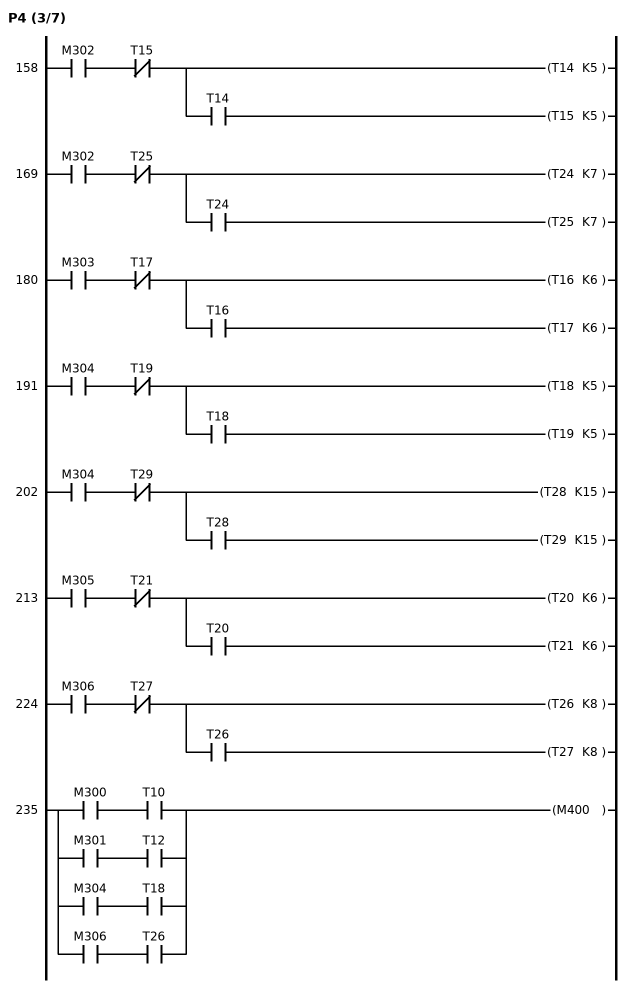
[picture p24: ladder of P4, rungs at steps 158 to 235]
158   LD      M302
      ANI     T15
      OUT     T14 K5
      AND     T14
      OUT     T15 K5
169   LD      M302
      ANI     T25
      OUT     T24 K7
      AND     T24
      OUT     T25 K7
180   LD      M303
      ANI     T17
      OUT     T16 K6
      AND     T16
      OUT     T17 K6
191   LD      M304
      ANI     T19
      OUT     T18 K5
      AND     T18
      OUT     T19 K5
202   LD      M304
      ANI     T29
      OUT     T28 K15
      AND     T28
      OUT     T29 K15
213   LD      M305
      ANI     T21
      OUT     T20 K6
      AND     T20
      OUT     T21 K6
224   LD      M306
      ANI     T27
      OUT     T26 K8
      AND     T26
      OUT     T27 K8
235   LD      M300
      AND     T10
      LD      M301
      AND     T12
      ORB
      LD      M304
      AND     T18
      ORB
      LD      M306
      AND     T26
      ORB
      OUT     M400
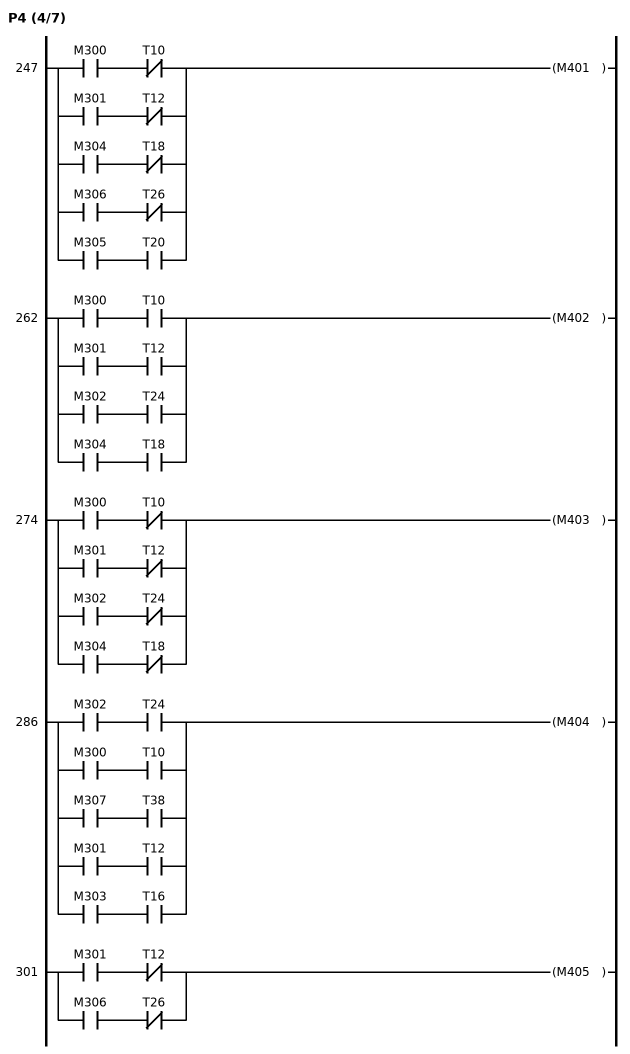
247   LD      M300
      ANI     T10
      LD      M301
      ANI     T12
      ORB
      LD      M304
      ANI     T18
      ORB
      LD      M306
      ANI     T26
      ORB
      LD      M305
      AND     T20
      ORB
      OUT     M401
262   LD      M300
      AND     T10
      LD      M301
      AND     T12
      ORB
      LD      M302
      AND     T24
      ORB
      LD      M304
      AND     T18
      ORB
      OUT     M402
274   LD      M300
      ANI     T10
      LD      M301
      ANI     T12
      ORB
      LD      M302
      ANI     T24
      ORB
      LD      M304
      ANI     T18
      ORB
      OUT     M403
286   LD      M302
      AND     T24
      LD      M300
      AND     T10
      ORB
      LD      M307
      AND     T38
      ORB
      LD      M301
      AND     T12
      ORB
      LD      M303
      AND     T16
      ORB
      OUT     M404
301   LD      M301
      ANI     T12
      LD      M306
      ANI     T26
      ORB
      OUT     M405
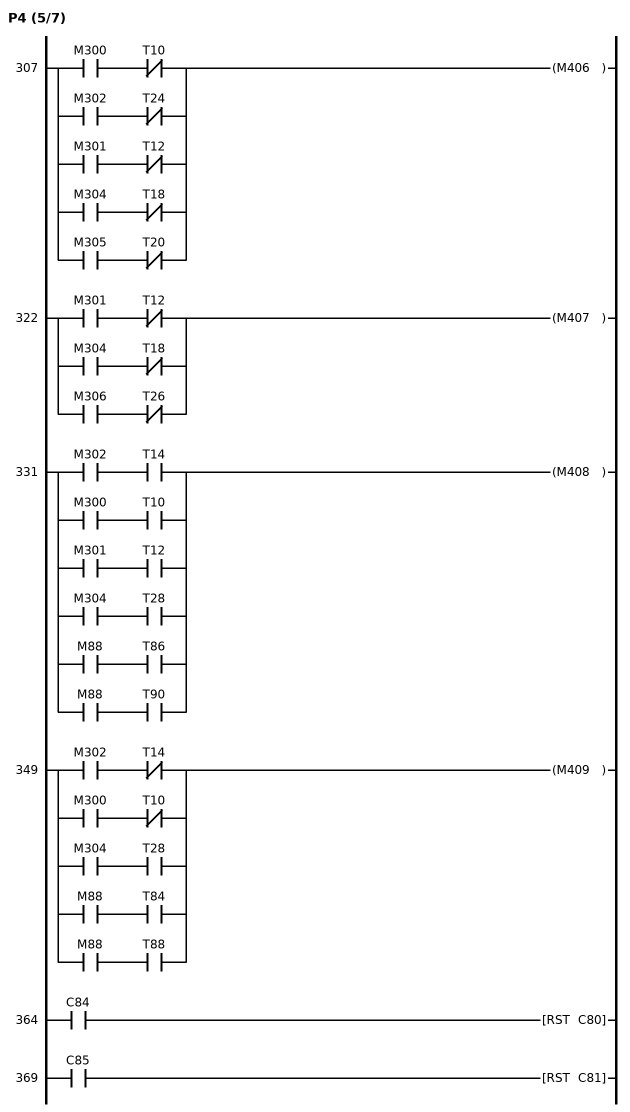
307   LD      M300
      ANI     T10
      LD      M302
      ANI     T24
      ORB
      LD      M301
      ANI     T12
      ORB
      LD      M304
      ANI     T18
      ORB
      LD      M305
      ANI     T20
      ORB
      OUT     M406
322   LD      M301
      ANI     T12
      LD      M304
      ANI     T18
      ORB
      LD      M306
      ANI     T26
      ORB
      OUT     M407
331   LD      M302
      AND     T14
      LD      M300
      AND     T10
      ORB
      LD      M301
      AND     T12
      ORB
      LD      M304
      AND     T28
      ORB
      LD      M88
      AND     T86
      ORB
      LD      M88
      AND     T90
      ORB
      OUT     M408
349   LD      M302
      ANI     T14
      LD      M300
      ANI     T10
      ORB
      LD      M304
      AND     T28
      ORB
      LD      M88
      AND     T84
      ORB
      LD      M88
      AND     T88
      ORB
      OUT     M409
364   LD      C84
      RST     C80
369   LD      C85
      RST     C81
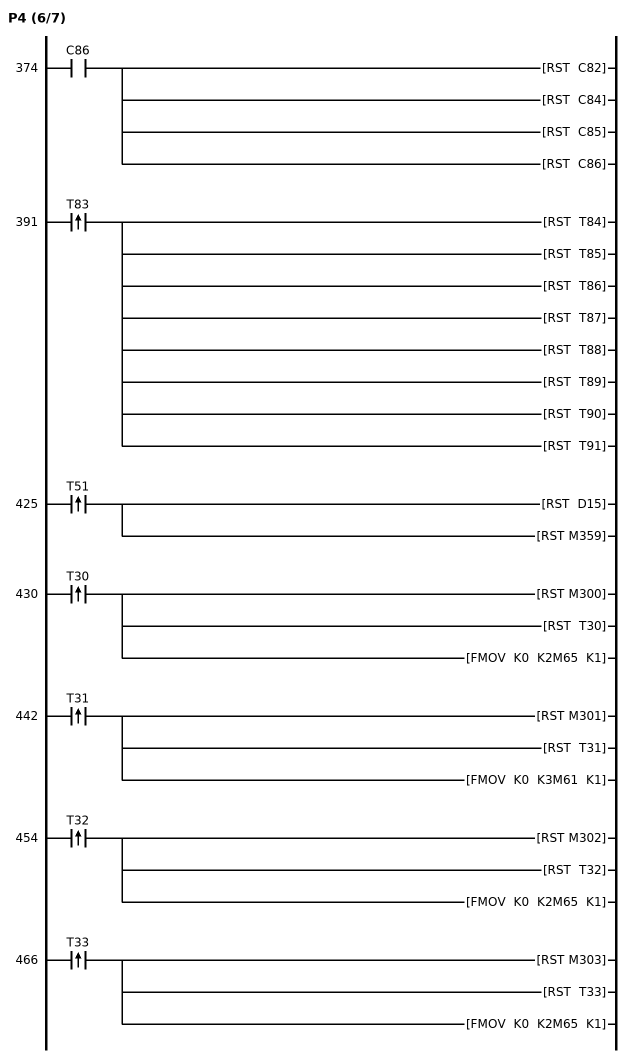
374   LD      C86
      RST     C82
      RST     C84
      RST     C85
      RST     C86
391   LDP     T83
      RST     T84
      RST     T85
      RST     T86
      RST     T87
      RST     T88
      RST     T89
      RST     T90
      RST     T91
425   LDP     T51
      RST     D15
      RST     M359
430   LDP     T30
      RST     M300
      RST     T30
      FMOV    K0 K2M65 K1
442   LDP     T31
      RST     M301
      RST     T31
      FMOV    K0 K3M61 K1
454   LDP     T32
      RST     M302
      RST     T32
      FMOV    K0 K2M65 K1
466   LDP     T33
      RST     M303
      RST     T33
      FMOV    K0 K2M65 K1
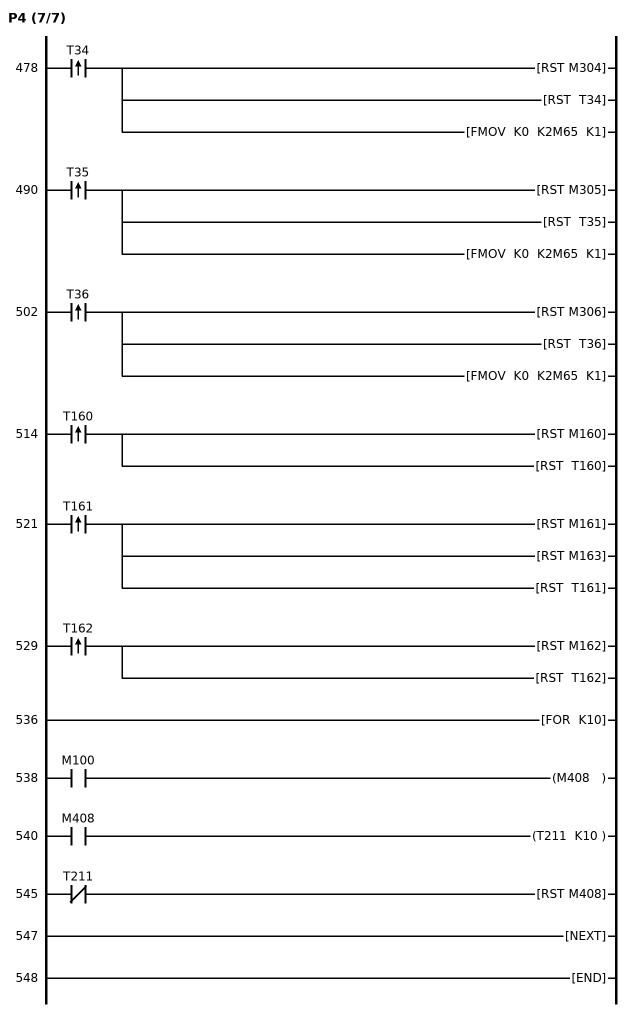
478   LDP     T34
      RST     M304
      RST     T34
      FMOV    K0 K2M65 K1
490   LDP     T35
      RST     M305
      RST     T35
      FMOV    K0 K2M65 K1
502   LDP     T36
      RST     M306
      RST     T36
      FMOV    K0 K2M65 K1
514   LDP     T160
      RST     M160
      RST     T160
521   LDP     T161
      RST     M161
      RST     M163
      RST     T161
529   LDP     T162
      RST     M162
      RST     T162
536   FOR     K10
538   LD      M100
      OUT     M408
540   LD      M408
      OUT     T211 K10
545   LDI     T211
      RST     M408
547   NEXT
548   END
END_PROGRAM

PROGRAM P5
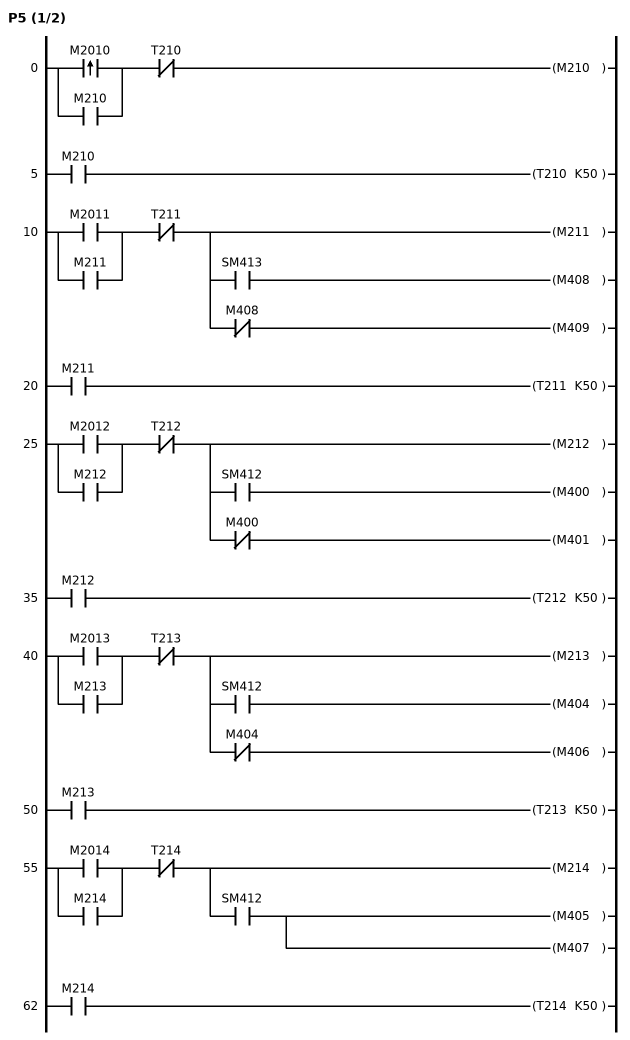
0     LDP     M2010
      OR      M210
      ANI     T210
      OUT     M210
5     LD      M210
      OUT     T210 K50
10    LD      M2011
      OR      M211
      ANI     T211
      OUT     M211
      MPS
      AND     SM413
      OUT     M408
      MPP
      ANI     M408
      OUT     M409
20    LD      M211
      OUT     T211 K50
25    LD      M2012
      OR      M212
      ANI     T212
      OUT     M212
      MPS
      AND     SM412
      OUT     M400
      MPP
      ANI     M400
      OUT     M401
35    LD      M212
      OUT     T212 K50
40    LD      M2013
      OR      M213
      ANI     T213
      OUT     M213
      MPS
      AND     SM412
      OUT     M404
      MPP
      ANI     M404
      OUT     M406
50    LD      M213
      OUT     T213 K50
55    LD      M2014
      OR      M214
      ANI     T214
      OUT     M214
      AND     SM412
      OUT     M405
      OUT     M407
62    LD      M214
      OUT     T214 K50
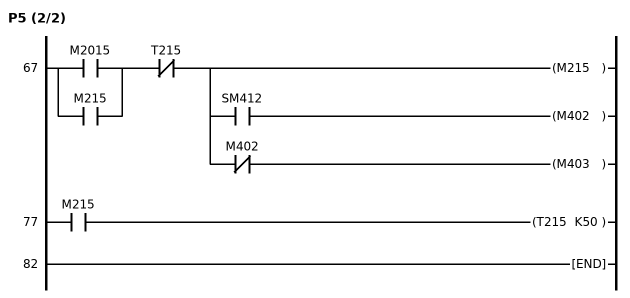
67    LD      M2015
      OR      M215
      ANI     T215
      OUT     M215
      MPS
      AND     SM412
      OUT     M402
      MPP
      ANI     M402
      OUT     M403
77    LD      M215
      OUT     T215 K50
82    END
END_PROGRAM

PROGRAM P6
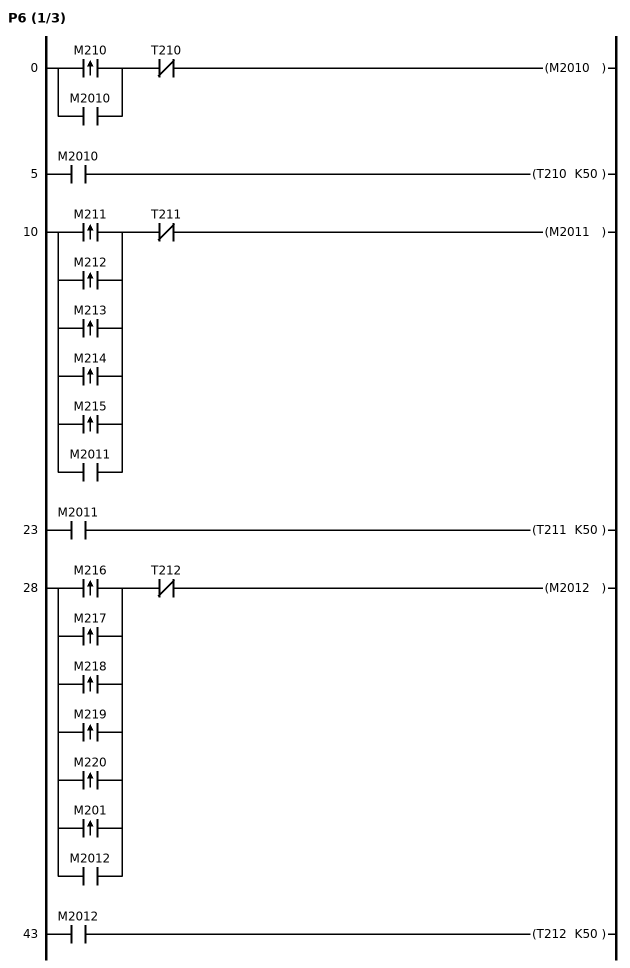
0     LDP     M210
      OR      M2010
      ANI     T210
      OUT     M2010
5     LD      M2010
      OUT     T210 K50
10    LDP     M211
      ORP     M212
      ORP     M213
      ORP     M214
      ORP     M215
      OR      M2011
      ANI     T211
      OUT     M2011
23    LD      M2011
      OUT     T211 K50
28    LDP     M216
      ORP     M217
      ORP     M218
      ORP     M219
      ORP     M220
      ORP     M201
      OR      M2012
      ANI     T212
      OUT     M2012
43    LD      M2012
      OUT     T212 K50
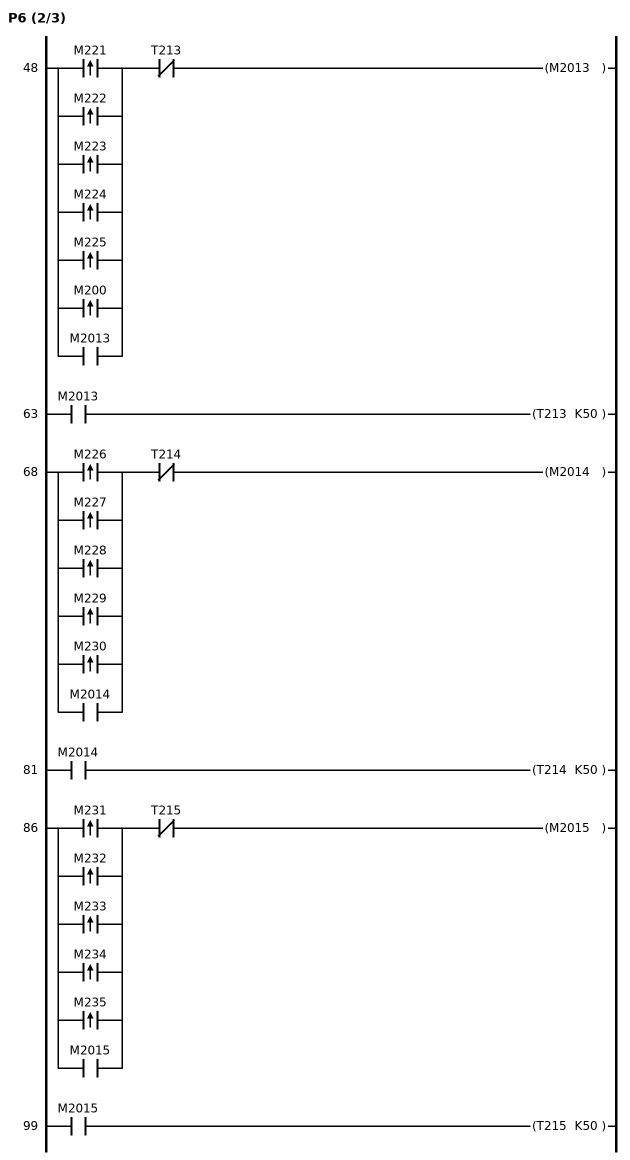
48    LDP     M221
      ORP     M222
      ORP     M223
      ORP     M224
      ORP     M225
      ORP     M200
      OR      M2013
      ANI     T213
      OUT     M2013
63    LD      M2013
      OUT     T213 K50
68    LDP     M226
      ORP     M227
      ORP     M228
      ORP     M229
      ORP     M230
      OR      M2014
      ANI     T214
      OUT     M2014
81    LD      M2014
      OUT     T214 K50
86    LDP     M231
      ORP     M232
      ORP     M233
      ORP     M234
      ORP     M235
      OR      M2015
      ANI     T215
      OUT     M2015
99    LD      M2015
      OUT     T215 K50
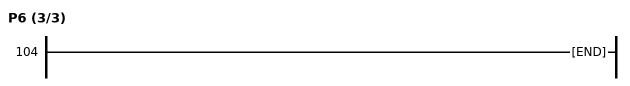
104   END
END_PROGRAM
